// TIA Portal V18 export
DATA_BLOCK "Parameters"   // DB1
{ S7_Optimized_Access := 'FALSE' }
VERSION : 0.1
// stored: AutoNumber true, IsOnlyStoredInLoadMemory false, IsWriteProtectedInAS false
   VAR RETAIN
      "Brakes On Time" : Time := T#500MS;
      "Brakes Off Time in Slow Mode" : Time := T#1S;
      "Brakes Off Time in Slow" : Time := T#200MS;
      "Brakes Off Time in Normal" : Time := T#800MS;
      "Cabin Driver Speed" : Int := 15000;
      "Canopy Up Timer" : Time := T#28S;
      "Cabin Motor Brake TOF" : Time := T#100MS;
      "Cab Angle Min" : Int := 7400;   // PBB1: -770, 19518, 0, 90, 0, 120 en sol
      "Cab Angle Max" : Int := 16500;
      "Cab Angle Min deg" : Real := 0.0;
      "Cab Angle Max deg" : Real := 135.0;
      "Cabin Stop Point Left" : Real := 0.1;
      "Cabin Stop Point Right" : Real := 135.0;
      "Drive Angle NomScale_test" : Real := 0.5;   // Ekrana sabit açı vermesi için. Test amaçlı
      "Drive Angle Min" : Int := 11750;
      "Drive Angle Max" : Int := 24000;
      "Drive Angle Min deg" : Real := 0.0;
      "Drive Angle Max deg" : Real := 180.0;
      "Drive Stop Point Left" : Real := 2.0;
      "Drive Stop Point Right" : Real := 178.0;
      "Drive Unit Stop-Slow Dif" : Real := 4.5;
      "Inclanation Desire Floor Point" : Real := 0.0;
      "Inclanation Auto Floor +- Tolerance" : Real := 0.0;
      "Laser Scale Min" : Int := 1000;
      "Laser Scale Max" : Int := 18000;
      "Laser Scale Min m" : Real := 23.5;
      "Laser Scale Max m" : Real := 36.2;
      "Laser FW Slow Point" : Real := 34.0;
      "Laser BW Slow Point" : Real := 25.0;
      "Laser FW Stop Point" : Real := 36.0;
      "Laser BW Stop Point" : Real := 23.5;
      "Laser FW Em Stop Point" : Real := 36.5;   // IPTAL
      "Laser BW Em Stop Point" : Real := 23.0;   // IPTAL
      "AutoLeveler Over Up Time" : Time := T#6S;
      "AutoLeveler Over Down Time" : Time := T#3S_500MS;
      "PBB Column Length" : Real := 5.67;
      "PBB Stop Point Up" : Real := 5.1;
      "PBB Stop Point Down" : Real := 1.8;
      "Rot Angle Min" : Int := 19850;
      "Rot Angle Max" : Int := 25850;
      "Rot Angle Min deg" : Real := 0.0;
      "Rot Angle Max deg" : Real := 180.0;
      "Rotunda Slow Point Right" : Real := 130.0;
      "Rotunda Slow Point LFT" : Real := 2.0;
      "Rotunda Stop Point Right" : Real := 135.0;
      "Rotunda Stop Point Left" : Real := 1.0;
      "Static_1 Time" : Time := T#0MS;
      "SafetyShoe Work Time" : Time := T#1S_500MS;
      "Slope Angle Min" : Real := 0.01;
      "Slope Angle Max" : Real := 7.5;
      "Slope Height Min" : Int := 0;   // PBB6:20625
      "Slope Height Max" : Int := 0;   // PBB6:17150
      "Slope Height Min m" : Real := 0.0;   // PBB6:1.57
      "Slope Height Max m" : Real := 0.0;   // PBB6:2.9
      "Slope Stop Point Max" : Real := 6.45;
      "Slope Stop Point Min" : Real := 0.1;
      "Slope Slow Point Max" : Real := 5.5;
      "Slope Slow Point Min" : Real := 0.05;
      "Speed Level 4" : Int := 4000;
      "Speed Level 1" : Int := 4000;
      "Speed Level 2" : Int := 8000;
      "Speed Level 3" : Int := 10000;
      "Wire Draw Min" : Int := 605;
      "Wire Draw Max" : Int := 15500;
      "Wire Draw Min M" : Real := 1.8;
      "Wire Draw Max M" : Real := 5.1;
      HmiDAY : Int := 29;
      HMI_MONTH : Int := 11;
      HMI_YEAR : Int := 2024;
      HMI_HOUR : Int := 15;
      HMI_MINUTE : Int := 7;
      "PLC_DAY_Set Point" : DTL := DTL#2024-08-05-00:00:00;
      HMI_DAY : DTL := DTL#2024-11-29-00:00:00;
      PLC_DAY_STOP : Bool := FALSE;
      "HMI Work Off Time" : Time := T#20M;
      "PBB Home position" : Real := 25.0;
   END_VAR
BEGIN
END_DATA_BLOCK
